       //Ir a Floor 3
       IF "posFloor3" = FALSE AND "send3Master" = TRUE AND "Var".MasterSendTo3 = FALSE THEN
           "slow" := FALSE;
           "toZ-" := FALSE;
           "toZ+" := FALSE;
           "Var".MasterSendTo3B2 := FALSE;
           "Var".MasterSendTo3B := FALSE;
           "Var".MasterSendTo3 := TRUE;
           "Var".MasterSendTo1 := FALSE;
           "Var".MasterSendTo1B := FALSE;
           "Var".MasterSendTo1B2 := FALSE;
           "Var".MasterSendTo2 := FALSE;
           "Var".MasterSendTo2B := FALSE;
           "Var".MasterSendTo2B2 := FALSE;
           "Var".MasterSendToGround := FALSE;
           "Var".MasterSendToGroundB := FALSE;
           "Var".MasterSendToGroundB2 := FALSE;
           "sendToGroundMaster" := FALSE;
           "sendTo1Master" := FALSE;
           "sendTo2Master" := FALSE;
           "sendTo3Master" := FALSE;
       END_IF;
       IF "Var".MasterSendTo3 = TRUE THEN
           IF "Var".MasterSendTo3B = FALSE THEN
               "Var".MasterSendTo3B := TRUE;
               "toZ+" := TRUE;
               "sendTo3Master" := TRUE;
           END_IF;
           IF "Var".MasterSendTo3B = TRUE AND "toZ+" = TRUE AND "slow3" = TRUE AND "slow" = FALSE THEN
               "Var".MasterSendTo3B := FALSE;
               "Var".MasterSendTo3B2 := TRUE;
               "slow" := TRUE;
           END_IF;
           IF "posFloor3" = TRUE THEN
               "slow" := FALSE;
               "toZ+" := FALSE;
               "Var".MasterSendTo3B2 := FALSE;
               "Var".MasterSendTo3B := FALSE;
               "Var".MasterSendTo3 := FALSE;
               "sendTo3Master" := FALSE;
           END_IF;
       END_IF;

       //Ir a Floor 1
       IF "posFloor1" = FALSE AND "send1Master" = TRUE AND "Var".MasterSendTo1 = FALSE THEN
           "slow" := FALSE;
           "toZ-" := FALSE;
           "toZ+" := FALSE;
           "Var".MasterSendTo3B2 := FALSE;
           "Var".MasterSendTo3B := FALSE;
           "Var".MasterSendTo3 := FALSE;
           "Var".MasterSendTo1 := TRUE;
           "Var".MasterSendTo1B := FALSE;
           "Var".MasterSendTo1B2 := FALSE;
           "Var".MasterSendTo2 := FALSE;
           "Var".MasterSendTo2B := FALSE;
           "Var".MasterSendTo2B2 := FALSE;
           "Var".MasterSendToGround := FALSE;
           "Var".MasterSendToGroundB := FALSE;
           "Var".MasterSendToGroundB2 := FALSE;
           "sendToGroundMaster" := FALSE;
           "sendTo1Master" := FALSE;
           "sendTo2Master" := FALSE;
           "sendTo3Master" := FALSE;
       END_IF;
       IF "Var".MasterSendTo1 = TRUE THEN
           IF ("floorIndicatorG" = TRUE AND "Var".MasterSendTo1B = FALSE) OR ("floorIndicator1" = TRUE AND "tempFloor2" = TRUE AND "Var".MasterSendTo1B = FALSE) THEN
               "Var".MasterSendTo1B := TRUE;
               "toZ+" := TRUE;
               "sendTo1Master" := TRUE;
           END_IF;
           IF "Var".MasterSendTo1B = TRUE AND "toZ+" = TRUE AND "slowBottom1" = TRUE AND "slow" = FALSE THEN
               "Var".MasterSendTo1B := FALSE;
               "slow" := TRUE;
           END_IF;
           IF (("floorIndicator2" = TRUE OR "floorIndicator3" = TRUE) AND "Var".MasterSendTo1B2 = FALSE) OR ("floorIndicator1" = TRUE AND "tempFloor4" = TRUE AND "Var".MasterSendTo1B2 = FALSE) THEN
               "Var".MasterSendTo1B2 := TRUE;
               "toZ-" := TRUE;
               "sendTo1Master" := TRUE;
           END_IF;
           IF "Var".MasterSendTo1B2 = TRUE AND "toZ-" = TRUE AND "slowTop1" = TRUE AND "slow" = FALSE THEN
               "Var".MasterSendTo1B2 := FALSE;
               "slow" := TRUE;
           END_IF;

           IF "posFloor1" = TRUE THEN
               "slow" := FALSE;
               "toZ+" := FALSE;
               "toZ-" := FALSE;
               "Var".MasterSendTo1B2 := FALSE;
               "Var".MasterSendTo1B := FALSE;
               "Var".MasterSendTo1 := FALSE;
               "sendTo1Master" := FALSE;
           END_IF;
       END_IF;

       //Ir a Floor 2
       IF "posFloor2" = FALSE AND "send2Master" = TRUE AND "Var".MasterSendTo2 = FALSE THEN
           "slow" := FALSE;
           "toZ-" := FALSE;
           "toZ+" := FALSE;
           "Var".MasterSendTo3B2 := FALSE;
           "Var".MasterSendTo3B := FALSE;
           "Var".MasterSendTo3 := FALSE;
           "Var".MasterSendTo1 := FALSE;
           "Var".MasterSendTo1B := FALSE;
           "Var".MasterSendTo1B2 := FALSE;
           "Var".MasterSendTo2 := TRUE;
           "Var".MasterSendTo2B := FALSE;
           "Var".MasterSendTo2B2 := FALSE;
           "Var".MasterSendToGround := FALSE;
           "Var".MasterSendToGroundB := FALSE;
           "Var".MasterSendToGroundB2 := FALSE;
           "sendToGroundMaster" := FALSE;
           "sendTo1Master" := FALSE;
           "sendTo2Master" := FALSE;
           "sendTo3Master" := FALSE;
       END_IF;
       IF "Var".MasterSendTo2 = TRUE THEN
           IF (("floorIndicatorG" = TRUE OR "floorIndicator1" = TRUE) AND "Var".MasterSendTo2B = FALSE) OR ("floorIndicator2" = TRUE AND "tempFloor5" = TRUE AND "Var".MasterSendTo2B = FALSE)  THEN
               "Var".MasterSendTo2B := TRUE;
               "toZ+" := TRUE;
               "sendTo2Master" := TRUE;
           END_IF;
           IF "Var".MasterSendTo2B = TRUE AND "toZ+" = TRUE AND "slowBottom2" = TRUE AND "slow" = FALSE THEN
               "Var".MasterSendTo2B := FALSE;
               "slow" := TRUE;
           END_IF;
           IF ("floorIndicator3" = TRUE AND "Var".MasterSendTo2B2 = FALSE) OR ("floorIndicator2" = TRUE AND "tempFloor7" = TRUE AND "Var".MasterSendTo2B2 = FALSE) THEN
               "Var".MasterSendTo2B2 := TRUE;
               "toZ-" := TRUE;
               "sendTo2Master" := TRUE;
           END_IF;
           IF "Var".MasterSendTo2B2 = TRUE AND "toZ-" = TRUE AND "slowTop2" = TRUE AND "slow" = FALSE THEN
               "Var".MasterSendTo2B2 := FALSE;
               "slow" := TRUE;
           END_IF;

           IF "posFloor2" = TRUE THEN
               "slow" := FALSE;
               "toZ+" := FALSE;
               "toZ-" := FALSE;
               "Var".MasterSendTo2B2 := FALSE;
               "Var".MasterSendTo2B := FALSE;
               "Var".MasterSendTo2 := FALSE;
               "sendTo2Master" := FALSE;
           END_IF;
       END_IF;

       //Alerta Master
       IF "alertMaster" = FALSE AND "Var".MasterAlertaB1 = FALSE AND "Var".MasterAlertaB2 = FALSE AND "Var".MasterAlertaB3 = FALSE THEN
           "alertIndMaster" := FALSE;
       END_IF;
       IF "alertMaster" = TRUE AND "alertIndMaster" = FALSE AND "Var".MasterAlertaB2 = FALSE AND "Var".MasterAlertaB3 = FALSE THEN
           "Var".MasterAlertaB1 := TRUE;
           "Var".MasterAlertaB2 := TRUE;
       END_IF;
       IF "Var".MasterAlertaB1 = TRUE AND "alertMaster" = FALSE AND "Var".MasterAlertaB2 = TRUE THEN
           "alertIndMaster" := TRUE;
           "Var".MasterAlertaB3 := TRUE;
       END_IF;
       IF "Var".MasterAlertaB1 = TRUE AND "alertMaster" = TRUE AND "Var".MasterAlertaB2 = TRUE AND "Var".MasterAlertaB3 = TRUE THEN
           "Var".MasterAlertaB1 := FALSE;
       END_IF;
       IF "Var".MasterAlertaB1 = FALSE AND "alertMaster" = FALSE AND "Var".MasterAlertaB2 = TRUE AND "Var".MasterAlertaB3 = TRUE THEN
           "alertIndMaster" := FALSE;
           "Var".MasterAlertaB2 := FALSE;
           "Var".MasterAlertaB3 := FALSE;
       END_IF;

       //Emergency Master
       IF "emergencyMaster" = FALSE AND "Var".MasterEmergencyB1 = FALSE AND "Var".MasterEmergencyB2 = FALSE AND "Var".MasterEmergencyB3 = FALSE THEN
           "emergencyIndMaster" := FALSE;
       END_IF;
       IF "emergencyMaster" = TRUE AND "emergencyIndMaster" = FALSE AND "Var".MasterEmergencyB2 = FALSE AND "Var".MasterEmergencyB3 = FALSE THEN
           "Var".MasterEmergencyB1 := TRUE;
           "Var".MasterEmergencyB2 := TRUE;
       END_IF;
       IF "Var".MasterEmergencyB1 = TRUE AND "emergencyMaster" = FALSE AND "Var".MasterEmergencyB2 = TRUE THEN
           "emergencyIndMaster" := TRUE;
           "Var".MasterEmergencyB3 := TRUE;
       END_IF;
       IF "Var".MasterEmergencyB1 = TRUE AND "emergencyMaster" = TRUE AND "Var".MasterEmergencyB2 = TRUE AND "Var".MasterEmergencyB3 = TRUE THEN
           "Var".MasterEmergencyB1 := FALSE;
       END_IF;
       IF "Var".MasterEmergencyB1 = FALSE AND "emergencyMaster" = FALSE AND "Var".MasterEmergencyB2 = TRUE AND "Var".MasterEmergencyB3 = TRUE THEN
           "emergencyIndMaster" := FALSE;
           "Var".MasterEmergencyB2 := FALSE;
           "Var".MasterEmergencyB3 := FALSE;
       END_IF;

   END_IF;
END_REGION
END_ORGANIZATION_BLOCK

(* ===== HMI "HMI_RT_1" =====
system functions are stored by id; their names below are inferred from use
connection "HMI_Connection_1": ETHERNET, S7_1500_OMS

HMI tags "Default tag table"
   "toZ+" : Bool = PLC "toZ+" AT %Q0.0, 1 s
   "toZ-" : Bool = PLC "toZ-" AT %Q0.1, 1 s
   "floorIndicatorG" : Bool = PLC floorIndicatorG AT %Q2.1, 1 s
   "cabinUp" : Bool = PLC cabinUp AT %Q2.6, 1 s
   "cabinDown" : Bool = PLC cabinDown AT %Q2.5, 1 s
   "floorIndicator1" : Bool = PLC floorIndicator1 AT %Q2.2, 1 s
   "floorIndicator2" : Bool = PLC floorIndicator2 AT %Q2.3, 1 s
   "floorIndicator3" : Bool = PLC floorIndicator3 AT %Q2.4, 1 s
   "overloadInd" : Bool = PLC overloadInd AT %Q3.5, 1 s
   "callToGround" : Bool = PLC callToGround AT %Q1.3, 1 s
   "callToDown1" : Bool = PLC callToDown1 AT %Q1.4, 1 s
   "callTo3" : Bool = PLC callTo3 AT %Q2.0, 1 s
   "callToUp2" : Bool = PLC callToUp2 AT %Q1.7, 1 s
   "callToDown2" : Bool = PLC callToDown2 AT %Q1.6, 1 s
   "callToUp1" : Bool = PLC callToUp1 AT %Q1.5, 1 s
   "alertInd" : Bool = PLC alertInd AT %Q3.3, 1 s
   "emergencyInd" : Bool = PLC emergencyInd AT %Q3.4, 1 s
   "Var_SimuladorEstado1" : Bool = PLC "Var".SimuladorEstado1, 1 s
   "Var_SimuladorEstado2" : Bool = PLC "Var".SimuladorEstado2, 1 s
   "Var_SimuladorEstado3" : Bool = PLC "Var".SimuladorEstado3, 1 s
   "Var_SimuladorEstado4" : Bool = PLC "Var".SimuladorEstado4, 1 s
   "Var_SimuladorEstado5" : Bool = PLC "Var".SimuladorEstado5, 1 s
   "Var_SimuladorEstado6" : Bool = PLC "Var".SimuladorEstado6, 1 s
   "Var_SimuladorEstado7" : Bool = PLC "Var".SimuladorEstado7, 1 s
   "Var_SimuladorEstado8" : Bool = PLC "Var".SimuladorEstado8, 1 s

Template "Template_1" 800x480
   Button "Exit" at 720,420 size 78x58; TextOff 'Exit'; PictureOff "ExitRuntime_TP700_Comfort_TR"; PictureOn "ExitRuntime_TP700_Comfort_TR"
      on Release: StopRuntime(0)
   Button "Log on" at 640,420 size 78x58; TextOff 'Log on'; PictureOff "Login_TP700_Comfort_TR"; PictureOn "Login_TP700_Comfort_TR"
      on Release: function_a2a04561()
   Button "Language" at 560,420 size 78x58; TextOff 'Language'; PictureOff "ToggleLanguage_TP700_Comfort_TR"; PictureOn "ToggleLanguage_TP700_Comfort_TR"
      on Release: function_fb9197e8(-1)
   Button "Template_Button" at 480,420 size 78x58; TextOff 'Text'
   Button "Template_Button_1" at 400,420 size 78x58; TextOff 'Text'
   Button "Template_Button_2" at 321,420 size 78x58; TextOff 'Text'
   Button "Template_Button_3" at 241,420 size 78x58; TextOff 'Text'
   Button "Template_Button_4" at 161,420 size 78x58; TextOff 'Text'
   Button "Alarms" at 81,420 size 78x58; TextOff 'Alarms'; PictureOff "AlarmDisplay_TP700_Comfort_TR"; PictureOn "AlarmDisplay_TP700_Comfort_TR"
      on Release: function_ef3f5d25("Alarm window_Unacknowledged", -1)
   Button "Start screen" at 1,420 size 78x58; TextOff 'Start screen'; PictureOff "NavigateHome_TP700_Comfort_TR"; PictureOn "NavigateHome_TP700_Comfort_TR"
      on Release: ActivateScreen("Root screen", 0)

screen "Root screen" 800x480, template "Template_1"
   TextField "Text field_1" at 413,31 size 316x28; Text 'HMI SIMULADOR ELEVADOR'
   Circle "Circle_1" at 593,98 size 28x28
      Appearance <- "cabinUp"
   TextField "Text field_2" at 630,98 size 99x23; Text 'SUBIENDO'
   Circle "Circle_2" at 593,135 size 28x28
      Appearance <- "cabinDown"
   Circle "Circle_3" at 593,172 size 28x28
      Appearance <- "floorIndicatorG"
   Circle "Circle_4" at 593,211 size 28x28
      Appearance <- "floorIndicator1"
   Circle "Circle_5" at 593,248 size 28x28
      Appearance <- "floorIndicator2"
   Circle "Circle_6" at 593,287 size 28x28
      Appearance <- "floorIndicator3"
   Circle "Circle_7" at 593,321 size 28x28
      Appearance <- "overloadInd"
   TextField "Text field_3" at 630,137 size 91x23; Text 'BAJANDO'
   TextField "Text field_4" at 630,175 size 111x23; Text 'Planta Baja'
   TextField "Text field_5" at 630,211 size 110x23; Text 'Primer Piso'
   TextField "Text field_6" at 630,250 size 126x23; Text 'Segundo Piso'
   TextField "Text field_7" at 630,287 size 108x23; Text 'Tercer Piso'
   TextField "Text field_8" at 630,326 size 99x23; Text 'Sobrepeso'
   Circle "Circle_8" at 390,98 size 28x28
      Appearance <- "callTo3"
   TextField "Text field_9" at 427,98 size 114x23; Text 'Llamar a TP'
   Circle "Circle_9" at 390,135 size 28x28
      Appearance <- "callToUp2"
   Circle "Circle_10" at 390,172 size 28x28
      Appearance <- "callToDown2"
   Circle "Circle_11" at 390,211 size 28x28
      Appearance <- "callToUp1"
   Circle "Circle_12" at 390,248 size 28x28
      Appearance <- "callToDown1"
   Circle "Circle_13" at 390,287 size 28x28
      Appearance <- "callToGround"
   Circle "Circle_14" at 390,321 size 28x28
      Appearance <- "alertInd"
   TextField "Text field_10" at 427,137 size 91x23; Text 'Arriba SP'
   TextField "Text field_11" at 427,175 size 87x23; Text 'Abajo SP'
   TextField "Text field_12" at 427,211 size 92x23; Text 'Arriba PP'
   TextField "Text field_13" at 427,250 size 88x23; Text 'Abajo PP'
   TextField "Text field_14" at 427,287 size 114x23; Text 'Llamar a PB'
   TextField "Text field_15" at 427,321 size 70x23; Text 'Alarma'
   Circle "Circle_15" at 390,355 size 28x28
      Appearance <- "emergencyInd"
   TextField "Text field_16" at 427,355 size 103x23; Text 'Emergency'
   Rectangle "Rectangle_4" at 153,315 size 107x74
      Visibility <- "Var_SimuladorEstado2"
   Rectangle "Rectangle_5" at 153,224 size 107x74
      Visibility <- "Var_SimuladorEstado4"
   Rectangle "Rectangle_6" at 153,135 size 107x74
      Visibility <- "Var_SimuladorEstado6"
   Rectangle "Rectangle_7" at 153,46 size 107x74
      Visibility <- "Var_SimuladorEstado8"
   Rectangle "Rectangle_8" at 153,315 size 54x74
      Visibility <- "Var_SimuladorEstado1"
   Rectangle "Rectangle_9" at 207,315 size 54x74
      Visibility <- "Var_SimuladorEstado1"
   Rectangle "Rectangle_10" at 261,315 size 54x74
      Visibility <- "Var_SimuladorEstado2"
   Rectangle "Rectangle_11" at 99,315 size 54x74
      Visibility <- "Var_SimuladorEstado2"
   Rectangle "Rectangle_12" at 98,224 size 54x74
      Visibility <- "Var_SimuladorEstado4"
   Rectangle "Rectangle_13" at 260,224 size 54x74
      Visibility <- "Var_SimuladorEstado4"
   Rectangle "Rectangle_14" at 152,224 size 54x74
      Visibility <- "Var_SimuladorEstado3"
   Rectangle "Rectangle_15" at 206,224 size 54x74
      Visibility <- "Var_SimuladorEstado3"
   Rectangle "Rectangle_16" at 101,135 size 54x74
      Visibility <- "Var_SimuladorEstado6"
   Rectangle "Rectangle_17" at 260,135 size 54x74
      Visibility <- "Var_SimuladorEstado6"
   Rectangle "Rectangle_18" at 155,135 size 54x74
      Visibility <- "Var_SimuladorEstado5"
   Rectangle "Rectangle_19" at 209,135 size 54x74
      Visibility <- "Var_SimuladorEstado5"
   Rectangle "Rectangle_20" at 98,46 size 54x74
      Visibility <- "Var_SimuladorEstado8"
   Rectangle "Rectangle_21" at 260,46 size 54x74
      Visibility <- "Var_SimuladorEstado8"
   Rectangle "Rectangle_22" at 152,46 size 54x74
      Visibility <- "Var_SimuladorEstado7"
   Rectangle "Rectangle_23" at 206,46 size 54x74
      Visibility <- "Var_SimuladorEstado7"
*)

(* ===== HMI "HMI_RT_2" =====
system functions are stored by id; their names below are inferred from use
connection "HMI_Connection_2": ETHERNET, S7_1500_OMS

HMI tags "Default tag table"
   "sendTo3" : Bool = PLC sendTo3 AT %Q3.2, 1 s
   "sendTo2" : Bool = PLC sendTo2 AT %Q3.1, 1 s
   "sendTo1" : Bool = PLC sendTo1 AT %Q3.0, 1 s
   "sendToGround" : Bool = PLC sendToGround AT %Q2.7, 1 s
   "Var_MASTER" : Bool = PLC "Var".MASTER, 1 s
   "alertInd" : Bool = PLC alertInd AT %Q3.3, 1 s
   "emergencyInd" : Bool = PLC emergencyInd AT %Q3.4, 1 s
   "emergency" : Bool = PLC emergency AT %I4.5, 1 s
   "alert" : Bool = PLC alert AT %I4.4, 1 s
   "sendGround" : Bool = PLC sendGround AT %I4.0, 1 s
   "send1" : Bool = PLC send1 AT %I4.1, 1 s
   "send2" : Bool = PLC send2 AT %I4.2, 1 s
   "send3" : Bool = PLC send3 AT %I4.3, 1 s
   "Var_MASTERINDICATOR" : Bool = PLC "Var".MASTERINDICATOR, 1 s
   "send3Master" : Bool = PLC send3Master AT %M0.4, 1 s
   "send2Master" : Bool = PLC send2Master AT %M0.3, 1 s
   "send1Master" : Bool = PLC send1Master AT %M0.2, 1 s
   "sendGroundMaster" : Bool = PLC sendGroundMaster AT %M0.1, 1 s
   "alertMaster" : Bool = PLC alertMaster AT %M0.5, 1 s
   "emergencyMaster" : Bool = PLC emergencyMaster AT %M0.6, 1 s
   "abrirPuertasMaster" : Bool = PLC abrirPuertasMaster AT %M0.7, 1 s
   "cerrarPuertasMaster" : Bool = PLC cerrarPuertasMaster AT %M1.0, 1 s
   "sendTo3Master" : Bool = PLC sendTo3Master AT %M2.0, 1 s
   "sendTo2Master" : Bool = PLC sendTo2Master AT %M2.1, 1 s
   "sendTo1Master" : Bool = PLC sendTo1Master AT %M2.2, 1 s
   "sendToGroundMaster" : Bool = PLC sendToGroundMaster AT %M2.3, 1 s
   "alarmIndMaster" : Bool = PLC alertIndMaster AT %M2.4, 1 s
   "emergencyIndMaster" : Bool = PLC emergencyIndMaster AT %M2.5, 1 s

Template "Template_1" 800x480
   Button "Exit" at 720,420 size 78x58; TextOff 'Exit'; PictureOff "ExitRuntime_TP700_Comfort_TR"; PictureOn "ExitRuntime_TP700_Comfort_TR"
      on Release: StopRuntime(0)
   Button "Log on" at 640,420 size 78x58; TextOff 'Log on'; PictureOff "Login_TP700_Comfort_TR"; PictureOn "Login_TP700_Comfort_TR"
      on Release: function_a2a04561()
   Button "Language" at 560,420 size 78x58; TextOff 'Language'; PictureOff "ToggleLanguage_TP700_Comfort_TR"; PictureOn "ToggleLanguage_TP700_Comfort_TR"
      on Release: function_fb9197e8(-1)
   Button "Template_Button" at 480,420 size 78x58; TextOff 'Text'
   Button "Template_Button_1" at 400,420 size 78x58; TextOff 'Text'
   Button "Template_Button_2" at 321,420 size 78x58; TextOff 'Text'
   Button "Template_Button_3" at 241,420 size 78x58; TextOff 'Text'
   Button "Template_Button_4" at 161,420 size 78x58; TextOff 'Text'
   Button "Alarms" at 81,420 size 78x58; TextOff 'Alarms'; PictureOff "AlarmDisplay_TP700_Comfort_TR"; PictureOn "AlarmDisplay_TP700_Comfort_TR"
      on Release: function_ef3f5d25("Alarm window_Unacknowledged", -1)
   Button "Start screen" at 1,420 size 78x58; TextOff 'Start screen'; PictureOff "NavigateHome_TP700_Comfort_TR"; PictureOn "NavigateHome_TP700_Comfort_TR"
      on Release: ActivateScreen("Root screen", 0)

screen "Root screen" 800x480, template "Template_1"
   TextField "Text field_1" at 455,34 size 251x28; Text 'HMI PANEL ELEVADOR'
   Button "Button_1" at 116,95 size 31x30; TextOff 'Text'
      on Press: SetBit("send3Master")
      on Release: ResetBit("send3Master")
   TextField "Text field_2" at 164,95 size 74x23; Text '3. Floor'
   Circle "Circle_1" at 262,91 size 27x27
      Appearance <- "sendTo3Master"
   Button "Button_2" at 116,140 size 31x30; TextOff 'Text'
      on Press: SetBit("send2Master")
      on Release: ResetBit("send2Master")
   Button "Button_3" at 114,183 size 31x30; TextOff 'Text'
      on Press: SetBit("send1Master")
      on Release: ResetBit("send1Master")
   Button "Button_4" at 115,226 size 31x30; TextOff 'Text'
      on Release: ResetBit("sendGroundMaster")
      on Press: SetBit("sendGroundMaster")
   Button "Button_5" at 115,266 size 31x30; TextOff 'Text'
      on Press: SetBit("alertMaster")
      on Release: ResetBit("alertMaster")
   TextField "Text field_3" at 164,140 size 74x23; Text '2. Floor'
   TextField "Text field_4" at 164,184 size 74x23; Text '1. Floor'
   TextField "Text field_5" at 169,227 size 70x23; Text 'Ground'
   TextField "Text field_6" at 173,269 size 59x23; Text 'Alarm'
   Circle "Circle_2" at 262,136 size 27x27
      Appearance <- "sendTo2Master"
   Circle "Circle_3" at 262,179 size 27x27
      Appearance <- "sendTo1Master"
   Circle "Circle_4" at 262,223 size 27x27
      Appearance <- "sendToGroundMaster"
   Circle "Circle_5" at 262,264 size 27x27
      Appearance <- "alarmIndMaster"
   Button "Button_6" at 115,305 size 31x30; TextOff 'Text'
      on Press: SetBit("emergencyMaster")
      on Release: ResetBit("emergencyMaster")
   TextField "Text field_7" at 157,307 size 103x23; Text 'Emergency'
   Circle "Circle_6" at 262,305 size 27x27
      Appearance <- "emergencyIndMaster"
   TextField "Text field_8" at 498,102 size 153x23; Text 'MODO MAESTRO'
   Button "Button_7" at 551,133 size 31x30; TextOff 'Text'
      on Press: SetBit("Var_MASTER")
      on Release: ResetBit("Var_MASTER")
   TextField "Text field_9" at 501,170 size 160x42; Text 'MODO MAESTRO ACTIVADO'
   Circle "Circle_7" at 554,216 size 27x27
      Appearance <- "Var_MASTERINDICATOR"
   Button "Button_8" at 479,261 size 31x30; TextOff 'Text'
      on Press: SetBit("abrirPuertasMaster")
      on Release: ResetBit("abrirPuertasMaster")
   TextField "Text field_10" at 524,263 size 127x23; Text 'Abrir Puertas'
   Button "Button_9" at 479,305 size 31x30; TextOff 'Text'
      on Press: SetBit("cerrarPuertasMaster")
      on Release: ResetBit("cerrarPuertasMaster")
   TextField "Text field_11" at 524,309 size 139x23; Text 'Cerrar Puertas'
*)